Staubli VAL3: init.pgx

program init(tool x_tTool (dimensions=1))
begin
  //-----------------------------------------------------------------------
  //Header begin
  //Description of program
  //  库变量初始
  //Input parameters
  //
  //Output paramaters
  //
  //Example
  //  call init(tool,frame,trTrsfOut)
  //History
  //  Creation : 2012-06-11 - PF.Zhong
  //Header end
  //-----------------------------------------------------------------------

  link(fFrame1,world)
  tTool=x_tTool
  //pFrameRefPt[0]:原点
  //pFrameRefPt[1]:X方向点
  //pFrameRefPt[2]:Y方向点
  //  pFrameRefPt[0]=here(tTool,world)
  //  pFrameRefPt[1]=here(tTool,world)
  //  pFrameRefPt[2]=here(tTool,world)
  bFrameTeach=false
  //  bFrameSave=false
  bExit=false
end
